// TIA Portal V19 export
DATA_BLOCK "Config"   // DB106
// stored: MemoryReserve 100, Namespace Unit2.EM0
   VAR
      em { ExternalWritable := 'False'} : "LAF_typeEmConfiguration";   // Configuration of EM Parameters
   END_VAR
BEGIN
   em.referenceDesignator.parent := WSTRING#'U1';
   em.referenceDesignator.relative := WSTRING#'EM1';
END_DATA_BLOCK
